{attribute 'qualified_only'}
{attribute 'strict'}
TYPE E_LenzeJogFreq :
(
	F0HZ 	:= 0,
	F20HZ	:= 1,
	F30HZ	:= 2,
	F40HZ	:= 3
);
END_TYPE

(* stored: Version 1.1.0.1, ProductVersion 3.1.4024.15
   EnumerationTextList E_LenzeJogFreq: Id {081d3483-9327-4626-aec1-ffe7666e79e4} *)
